{attribute 'GeneratedUsingTerminal: EL1054-0000-0016'}
{attribute addProperty BoxType "EL1054-0000-0016"}
{attribute addProperty Description "EL1054 4Ch. Dig. Input, NAMUR sensors"}
{attribute addProperty Physics "KK"}
{attribute addProperty Id "Channel_1AT %I*Channel_31CEFA7F2Channel_2AT %I*Channel_31CEFA7F2Channel_3AT %I*Channel_31CEFA7F2Channel_4AT %I*Channel_31CEFA7F2WcStateAT %I*WcState_9091E0EB2InfoDataAT %I*InfoData_6F19DB2B2"}
{attribute addProperty CRC "935885340"}
{attribute addProperty Size "12"}
TYPE EL1054_37C87A1C EXTENDS EtcSlaveTerminalBase_947E5A46 :
STRUCT
	{attribute addProperty Name "Channel_1"}
	Channel_1 : Channel_31CEFA7F;
	{attribute addProperty Name "Channel_2"}
	Channel_2 : Channel_31CEFA7F;
	{attribute addProperty Name "Channel_3"}
	Channel_3 : Channel_31CEFA7F;
	{attribute addProperty Name "Channel_4"}
	Channel_4 : Channel_31CEFA7F;
	{attribute addProperty Name "WcState"}
	WcState : WcState_9091E0EB;
	{attribute addProperty Name "InfoData"}
	InfoData : InfoData_6F19DB2B;
END_STRUCT
END_TYPE

(* stored: Version 1.2.0.0, ProductVersion 3.1.4024.9
   DUT EL1054_37C87A1C: Id {b4431b9c-968b-43ef-a145-da3dec76d025} *)
